screen "Symulacja_czujnikow" 800x480
   TextField "Text field_1" at 12,58 size 252x23; Text 'Czujnik Wilgotności powietrza'
   TextField "Text field_2" at 306,58 size 214x23; Text 'Czujnik Wilgotności gleby'
   TextField "Text field_3" at 32,202 size 202x23; Text 'Termometr wewnętrzny'
   TextField "Text field_4" at 323,202 size 197x23; Text 'Termometr zewnętrzny'
   TextField "Text field_5" at 566,58 size 216x23; Text 'Czujnik natężenia światła'
   TextField "Text field_6" at 607,202 size 124x23; Text 'Czujnik wiatru'
   TextField "Text field_7" at 27,346 size 208x23; Text 'Wewnętrzny czujnik CO2'
   TextField "Text field_8" at 306,346 size 202x23; Text 'Zewnętrzny czujnik CO2'
   TextField "Text field_9" at 569,346 size 206x23; Text 'Stopień zasłonięcia rolet'
   IOField "I/O field_4" at 599,94 size 150x60; FormatPattern 9999
      ProcessValue <- "Czujnik_natezenia_światła"
   IOField "I/O field_5" at 599,242 size 150x60; FormatPattern 999
      ProcessValue <- "Czujnik_wiatru"
   IOField "I/O field_6" at 69,375 size 150x60; FormatPattern 9999
      ProcessValue <- "Wewnetrzny_czujnik_CO2"
   IOField "I/O field_7" at 346,375 size 150x60; FormatPattern 9999
      ProcessValue <- "Zewnetrzny_czujnik_CO2"
   IOField "I/O field_8" at 599,375 size 150x60; FormatPattern 999
      ProcessValue <- "Stopien_zasloniecia_rolet"
   IOField "I/O field_10" at 69,94 size 150x60; FormatPattern 999
      ProcessValue <- "Czujnik_wilgotności_powietrza"
   IOField "I/O field_11" at 346,94 size 150x60; FormatPattern 999
      ProcessValue <- "Czujnik_wilgotności_gleby"
   IOField "I/O field_12" at 69,242 size 150x60; FormatPattern 99.9
      ProcessValue <- "Temperatura_wewnetrzna"
   IOField "I/O field_13" at 346,242 size 150x60; FormatPattern 99.9
      ProcessValue <- "Temperatura_zewnetrzna"
   TextField "Text field_10" at 248,5 size 321x34; Text 'ZAPISZ RECEPTURE / SYMULACJA CZUJNIKÓW'
   Button "Button_1" at 750,0 size 50x50; TextOff 'WRÓĆ'; PictureOff "Back_arrow"
      on Click: function_efd93a16()
   Button "Button_14" at 3,1 size 43x43; TextOff 'DOM'; PictureOff "home_1"
      on Click: ActivateScreen("Root screen", 0)

screen "tryb_automatyczny" 800x480
   on GenerateScreen: SetTag("Tag_ScreenNumber", 1)
   IOField "I/O field_1" at 67,322 size 57x40; FormatPattern 99.9
      ProcessValue <- "Temperatura_wewnetrzna"
   Button "Button_1" at 745,0 size 55x55; TextOff 'WRÓĆ'; PictureOff "Back_arrow"
      on Click: function_efd93a16()
   Button "Button_2" at 373,382 size 416x89; TextOff 'ZATWIERDŹ'
      on Click: ResetBit("HMI_Reset_Trybow"); SetBit("HMI_Aktywacja_trybu_automatycznego"); ActivateScreen("praca", 0)
   Bar "Bar_1" at 7,110 size 50x250; MinimumValue 0; MaximumValue 45
      ProcessValue <- "Temperatura_auto"
   TextField "Text field_2" at 1,71 size 132x23; Text 'TEMPERATURA'
   Bar "Bar_2" at 170,111 size 50x250; MinimumValue 0; MaximumValue 100
      ProcessValue <- "Wilgotnosc_powietrza_auto"
   TextField "Text field_3" at 165,68 size 122x42; Text 'WOLGOTNOŚĆ POWIETRZA WILGOTNOŚĆ POWIETRZA'
   Button "Button_3" at 71,115 size 75x45; TextOff '+ / +0.5 °C'
      on Press: function_dd21b452("Temperatura_auto", 0.5)
   Button "Button_7" at 71,183 size 75x45; TextOff '- / -0.5 °C'
      on Press: function_b9b71300("Temperatura_auto", 0.5)
   IOField "I/O field_2" at 67,251 size 62x40; FormatPattern 99.9
      ProcessValue <- "Temperatura_auto"
   TextField "Text field_11" at 122,260 size 23x22; Text '°C'
   TextField "Text field_9" at 122,333 size 23x22; Text '°C'
   Bar "Bar_4" at 335,111 size 50x250; MinimumValue 0; MaximumValue 100
      ProcessValue <- "Wilgotnosc_gleby_auto"
   TextField "Text field_10" at 332,65 size 122x42; Text 'WOLGOTNOŚĆ GLEBY WILGOTNOŚĆ GLEBY'
   Button "Button_8" at 398,132 size 65x40; TextOff '+ / +2%'
      on Click: function_dd21b452("Wilgotnosc_gleby_auto", 2)
   Button "Button_9" at 398,181 size 65x40; TextOff '- / -2%'
      on Click: function_b9b71300("Wilgotnosc_gleby_auto", 2)
   IOField "I/O field_5" at 402,255 size 60x40; FormatPattern 999
      ProcessValue <- "Wilgotnosc_gleby_auto"
   IOField "I/O field_6" at 404,325 size 58x40; FormatPattern 999
      ProcessValue <- "Czujnik_wilgotności_gleby"
   TextField "Text field_12" at 385,243 size 101x22; Text 'USTAWIONA'
   TextField "Text field_13" at 389,314 size 86x22; Text 'AKTUALNA'
   TextField "Text field_14" at 439,264 size 23x22; Text '%'
   TextField "Text field_15" at 439,335 size 23x22; Text '%'
   Button "Button_10" at 229,126 size 65x40; TextOff '+ / +5%'
      on Click: function_dd21b452("Wilgotnosc_powietrza_auto", 5)
   Button "Button_11" at 229,186 size 65x40; TextOff '- / -5%'
      on Click: function_b9b71300("Wilgotnosc_powietrza_auto", 5)
   IOField "I/O field_4" at 234,248 size 66x40; FormatPattern 999
      ProcessValue <- "Wilgotnosc_powietrza_auto"
   IOField "I/O field_7" at 236,320 size 62x40; FormatPattern 999
      ProcessValue <- "Czujnik_wilgotności_powietrza"
   TextField "Text field_16" at 223,235 size 101x22; Text 'USTAWIONA'
   TextField "Text field_17" at 223,306 size 86x22; Text 'AKTUALNA'
   TextField "Text field_18" at 275,257 size 23x22; Text '%'
   TextField "Text field_19" at 275,328 size 23x22; Text '%'
   Button "Button_14" at 4,7 size 45x45; TextOff 'DOM'; PictureOff "home_1"
      on Click: ActivateScreen("Root screen", 0)
   TextField "Text field_4" at 143,381 size 128x23; Text 'SYSTEM OKIEN'
   Switch "Switch_1" at 106,410 size 216x46; TextOn 'ON'; CaptionText 'Switch'; TextOff 'OFF'
      ProcessValue <- "System_okien_auto"
   GraphicView "Graphic view_1" at 129,70 size 40x40; Picture "Thermometer_icon"
   GraphicView "Graphic view_2" at 281,68 size 40x40; Picture "sensor_4212519"
   TextField "Text field_5" at 60,309 size 86x22; Text 'AKTUALNA'
   TextField "Text field_6" at 57,237 size 101x22; Text 'USTAWIONA'
   GraphicView "Graphic view_3" at 443,71 size 40x40; Picture "soil-sensor_11298794"
   TextField "Text field_1" at 255,4 size 291x47; Text 'TRYB AUTOMATYCZNY'
   Bar "Bar_3" at 496,111 size 50x250; MinimumValue 0; MaximumValue 1500
      ProcessValue <- "Naslonecznienie_auto"
   TextField "Text field_7" at 492,55 size 154x40; Text 'WOLGOTNOŚĆ GLEBY NASŁONECZNIENIE'
   GraphicView "Graphic view_4" at 585,86 size 40x40; Picture "sensor_4212513"
   Button "Button_4" at 553,131 size 82x43; TextOff '+ +50 W m'
      on Click: function_dd21b452("Naslonecznienie_auto", 50)
   Button "Button_5" at 554,186 size 82x43; TextOff '- -50 W m'
      on Click: function_b9b71300("Naslonecznienie_auto", 50)
   IOField "I/O field_3" at 561,254 size 61x40; FormatPattern 9999
      ProcessValue <- "Naslonecznienie_auto"
   TextField "Text field_8" at 545,242 size 101x22; Text 'USTAWIONA / USTAWIONE'
   IOField "I/O field_8" at 563,325 size 62x40; FormatPattern 9999
      ProcessValue <- "Czujnik_natezenia_światła"
   TextField "Text field_20" at 549,313 size 86x22; Text 'AKTUALNA / AKTUALNE'
   TextField "Text field_23" at 616,150 size 32x18; Text '2'
   TextField "Text field_24" at 614,205 size 32x18; Text '2'
   Bar "Bar_5" at 656,111 size 45x250; MinimumValue 400; MaximumValue 950
      ProcessValue <- "Poziom_CO2_auto"
   TextField "Text field_21" at 656,65 size 128x23; Text 'SYSTEM OKIEN / POZIOM CO2'
   IOField "I/O field_9" at 723,254 size 66x40; FormatPattern 999
      ProcessValue <- "Poziom_CO2_auto"
   TextField "Text field_22" at 699,216 size 101x22; Text 'USTAWIONA / USTAWIONE'
   IOField "I/O field_10" at 723,333 size 62x40; FormatPattern 999
      ProcessValue <- "Wewnetrzny_czujnik_CO2"
   TextField "Text field_25" at 708,314 size 86x22; Text 'AKTUALNA'
   Button "Button_6" at 714,134 size 73x40; TextOff '+ / +25ppm'
      on Click: function_dd21b452("Poziom_CO2_auto", 25)
   Button "Button_12" at 714,186 size 73x40; TextOff '+ / -25ppm'
      on Click: function_b9b71300("Poziom_CO2_auto", 25)
   GraphicView "Graphic view_5" at 754,83 size 40x40; Picture "sensor_2828470"
   GraphicView "Graphic view_6" at 17,400 size 55x55; Picture "window_11250237"
*)